// Miscellaneous.
FUNCTION_BLOCK FB_Misc EXTENDS FB_BA_View
VAR	
	// Intention:		Adjust certain ("BA_Param" related) settings via PLC code.
	//					> Feel free to implement as muss instances as needed, where ever needed.
	Settings			: FB_BA_Settings := (
							EventEn_Simple			:= F_BA_EventTransition(TRUE, FALSE, FALSE),
							EventEn_Standard		:= F_BA_EventTransition(TRUE, FALSE, FALSE),
							EventEn_Extended		:= F_BA_EventTransition(TRUE, FALSE, TRUE),
							EvtMgmt_AckMode			:= E_BA_AcknowledgeMode.eEntire,
							
							// Intention:			Adjust access to some specific parameters (Leaving rest untouched).
							DefWriteAccess			:= F_BA_ParameterRolesBuilder()
														.Set(E_BA_Parameter.eEventEnable, E_BA_Role.eInternal)
														.Build()
						);
							
	// Intention:		Initialize some special UTF-8 characters.
	SpecialUtf8			: FB_BA_AV_Op := (
							iParent					:= THIS^,
							sDescription			:= wsLiteral_TO_UTF8("{äöüßéèêµ€° Ἀθῆναι İstanbul Київ}"),
							eUnit					:= E_BA_Unit.eOther_Percent,
							fValueRm				:= 5
						);
END_VAR

SUPER^();

SpecialUtf8();

END_FUNCTION_BLOCK

(* stored: Version 1.1.0.1, ProductVersion 3.1.4024.9
   POU FB_Misc: Id {3ab59abd-7907-417e-9172-68b9f3ae54be}, SpecialFunc None *)
